(* PLC project Arbeitsmaschine7, KW-Software MULTIPROG 5.35 *)
(* stored: companyURL www.kw-software.com, productRelease Build 434, creationDateTime 2012-11-13T09:01:25, version 1352793685, modificationDateTime 2012-11-13T09:01:25 *)

(* Layer 3: Ablaufebene --> Greift auf Layer 2 zu. Der FB spiegelt die Funktion "Transport nach x, Bearbeitung" eines Werkstücks wider. Der Unterschied zum FB "Bearbeiten" aus Layer 2 besteht darin, dass der Bearbeitungsablauf neben dem reinen Bearbeiten des Werkstückes auch die Übernahme/Übergabe, das Transportieren des Werkstücks, die Werkzeugauswahl und die Höhenänderung des Werkzeugs umfasst. Die Ansteuerung der drei Transportzustände (nach links, nach rechts und aus) wird durch zwei Variablen (Transport_nach_links, Transport_nach_rechts) realisiert. Die Ansteuerung der 4 Bearbeitungszustände wird über 3 Variablen (Bearbeiten1, Bearbeiten2, Bearbeiten3) realisiert. Im Anfangsschritt findet keine Bearbeitung statt - kein Bearbeiten/Transportieren/Übergeben/Übernehmen/ Werkzeug auswählen/keine Höhenänderung (Motoren aus). Je nach Setzen der Inputvariablen (alternative Verzweigung) wird ein Werkstück von der entsprechenden Seite übernommen. Liefert FB "Übernahme_gabe" das Quittierungssignal, dass erfolgreich übernommen wurde, schaltet die Transition. Damit wird ein Zustand eingenommen, der erstmal alle Motoren stoppt (Wichtig ist, dass der Transportbandmotor gestoppt wird.). Nun wird entsprechend der Inputvariablen die Auwahl des Werkzeuges vorgenommen. Liefert der FB "Werkzeugauswahl" das Quittierungssignal, dass das Werkzeug erfolgreich ausgewählt wurde, dann schaltet die Transition. Nun wird geprüft, ob ein Verfahren des Werkzeuges nötig ist und das Werkzeug gegebenenfalls verfahren werden muss. Wurde das Werkzeug bereits auf die unterste Position verfahren, so ist kein weiteres Verfahren des Werkzeuges nötig. Ebenfalls ist ein Verfahren des Werkzeuges unnötig, wenn kein Werkstück zur Bearbeitung bereitliegt. Nach erfolgreichem Verfahren des Werkzeuges, liefert der FB "Werkzeughoehe" das Quittierungssignal und die Transition schaltet. Nun wird das Werkzeug entsprechend der Inputvariablen bearbeitet. Wenn die Bearbeitung abgeschlossen ist, wird vom FB "Bearbeiten" ein Quittierungssignal gesendet und die Transition schaltet. Nun wird geprüft, ob ein Verfahren des Werkzeuges nötig ist und das Werkzeug gegebenenfalls verfahren werden muss. Befindet sich das Werkzeug bereits auf der höhsten Position, so ist ein erneutes Verfahren des Werkzeugs nicht nötig. Nach erfolgreichem Verfahren des Werkzeuges liefert der FB "Werkzeughoehe" das Quittierungssignal und die Transition schaltet. Nun schaltet die Transition "T_XXX_ein" und das Werkstück wird in die entsprechende Richtung transportiert. Liefert FB "Transportieren" das Quittierungssignal, dass erfolgreich transportiert wurde, schaltet die Transition. Damit wird ein Zustand eingenommen, der alle Motoren stoppt (Wichtig ist, dass der Transportbandmotor gestoppt wird.). Nach Auswertung der Bedingungen, an welcher Seite das Werkstück übergeben werden muss, wird der Zustand eingenommen,der das Werkstück übergibt. Wurde erfolgreich übergeben, so ist der Bearbeitungsablauf abgeschlossen. Dabei wird auch eine Statusvariable gesetzt (TPB_xxx), die den erfolgreichen Bearbeitungsablauf quittiert, sodass die übergeordnete Steuerung weiß, wann der Transportvorgang und der Bearbeitungsvorgang abgeschlossen ist. FB-Schnittstellen: --------------- Eingangsvariablen: - Bearbeiten1 - Bearbeiten2 - Bearbeiten3 - Transport_nach_links - Transport_nach_rechts Ausgangsvariablen: - TPB_links - TPB_rechts Auftretende Warnungen "Instanz 'FB_xxx' mehrfach verwendet!": Hier ein Textauszug aus der Multiprog-Hilfe: "Die Warnung kann auch in einem Code-Arbeitsblatt in AS auftreten, wenn Sie dieselbe Instanz in verschiedenen Aktionen verwendet haben. Wenn nur eine Instanz zu einem Zeitpunkt ausgeführt wird, ist die Warnung für Sie ohne Bedeutung." *)
FUNCTION_BLOCK Transport_zu_x_Bearbeit
  VAR
    FB_Uebergabe : Uebernahme_gabe;
    FB_Uebernahme : Uebernahme_gabe;
    FB_Bearbeiten : Bearbeiten;
    FB_Werkzeugauswahl : Werkzeugauswahl;
    FB_Werkzeughoehe : Werkzeughoehe;
  END_VAR
  VAR_INPUT
    Transport_nach_links : BOOL := FALSE;
    Transport_nach_rechts : BOOL := FALSE;
  END_VAR
  VAR
    Quittierungssignal_links1 : BOOL := FALSE;
    Quittierungssignal_rechts1 : BOOL := FALSE;
    Quittierungssignal_links2 : BOOL := FALSE;
    Quittierungssignal_rechts2 : BOOL := FALSE;
  END_VAR
  VAR_INPUT
    Bearbeiten1 : BOOL := FALSE;
    Bearbeiten2 : BOOL := FALSE;
    Bearbeiten3 : BOOL := FALSE;
  END_VAR
  VAR
    Sensor_Auswahl : BOOL := FALSE;
    links : BOOL := FALSE;
    rechts : BOOL := FALSE;
    Quittierungssignal_Wahl1 : BOOL := FALSE;
    Quittierungssignal_Wahl2 : BOOL := FALSE;
    Quittierungssignal_Wahl3 : BOOL := FALSE;
    Quittierungssignal_ab : BOOL := FALSE;
    Hoehe_0 : BOOL := FALSE;
    Quittierungssignal_WZ1 : BOOL := FALSE;
    Quittierungssignal_WZ2 : BOOL := FALSE;
    Quittierungssignal_WZ3 : BOOL := FALSE;
    Quittierungssignal_auf : BOOL := FALSE;
    Quittierungssignal_links3 : BOOL := FALSE;
    Quittierungssignal_rechts3 : BOOL := FALSE;
    Quittierungssignal_links4 : BOOL := FALSE;
    Quittierungssignal_rechts4 : BOOL := FALSE;
  END_VAR
  VAR_OUTPUT
    TPB_rechts : BOOL := FALSE;
    TPB_links : BOOL := FALSE;
  END_VAR
  VAR
    FB_Werkzeughoehe_auf : Werkzeughoehe;
    FB_Werkzeughoehe_ab : Werkzeughoehe;
    FB_Positionieren : Positionieren;
    Quittierungssignal_Pos_links : BOOL := FALSE;
    Quittierungssignal_Pos_rechts : BOOL := FALSE;
  END_VAR

(* transition T_Uebergeben_r_aus *)
FB_Uebergabe();
Quittierungssignal_rechts4 := FB_Uebergabe.UeG_UeN_rechts;
IF Quittierungssignal_rechts4 = TRUE
	THEN T_Uebergeben_r_aus := TRUE;
	ELSE T_Uebergeben_r_aus := FALSE;
END_IF;
(* transition T_Uebergeben_l_aus *)
FB_Uebergabe();
Quittierungssignal_links4 := FB_Uebergabe.UeG_UeN_links;
IF Quittierungssignal_links4 = TRUE
	THEN T_Uebergeben_l_aus := TRUE;
	ELSE T_Uebergeben_l_aus := FALSE;
END_IF;
(* transition T_Uebergeben_r_ein *)
FB_Uebernahme();
Quittierungssignal_rechts3 := FB_Uebernahme.UeG_UeN_rechts;
IF Quittierungssignal_rechts3 = TRUE
	THEN T_Uebergeben_r_ein := TRUE; 
	ELSE T_Uebergeben_r_ein := FALSE;
END_IF;
(* transition T_Uebergeben_l_ein *)
FB_Uebernahme();
Quittierungssignal_links3 := FB_Uebernahme.UeG_UeN_links;
IF Quittierungssignal_links3 = TRUE 
	THEN T_Uebergeben_l_ein := TRUE; 
	ELSE T_Uebergeben_l_ein := FALSE;
END_IF;
(* transition T_Hoehe_aufwaerts_aus *)
FB_Werkzeughoehe_auf();
Quittierungssignal_auf := FB_Werkzeughoehe_auf.Hoehe_auf;
IF Quittierungssignal_auf = TRUE
	THEN T_Hoehe_aufwaerts_aus := TRUE;
	ELSE T_Hoehe_aufwaerts_aus := FALSE;
END_IF;
(* transition T_keine_Hoehenaenderung2 *)
FB_Werkzeughoehe();
Hoehe_0 := FB_Werkzeughoehe.Position0;
IF Hoehe_0 = TRUE
	THEN T_keine_Hoehenaenderung2 := TRUE; 
	ELSE T_keine_Hoehenaenderung2 := FALSE;
END_IF;
(* transition T_Hoehe_aufwaerts_ein *)
FB_Werkzeughoehe();
Hoehe_0 := FB_Werkzeughoehe.Position0;
IF Hoehe_0 = FALSE
	THEN T_Hoehe_aufwaerts_ein := TRUE; 
	ELSE T_Hoehe_aufwaerts_ein := FALSE;
END_IF;
(* transition T_Werkzeug3_aus *)
FB_Bearbeiten();
Quittierungssignal_WZ3 := FB_Bearbeiten.BA_WZ3;
IF Quittierungssignal_WZ3 = TRUE
	THEN T_Werkzeug3_aus := TRUE;
	ELSE T_Werkzeug3_aus := FALSE;
END_IF;
(* transition T_Werkzeug2_aus *)
FB_Bearbeiten();
Quittierungssignal_WZ2 := FB_Bearbeiten.BA_WZ2;
IF Quittierungssignal_WZ2 = TRUE
	THEN T_Werkzeug2_aus := TRUE;
	ELSE T_Werkzeug2_aus := FALSE; 
END_IF;
(* transition T_Werkzeug1_aus *)
FB_Bearbeiten();
Quittierungssignal_WZ1 := FB_Bearbeiten.BA_WZ1;
IF Quittierungssignal_WZ1 = TRUE
	THEN T_Werkzeug1_aus := TRUE;
	ELSE T_Werkzeug1_aus := FALSE;
END_IF;
(* transition T_Werkzeug3_ein *)
IF Bearbeiten1 = FALSE AND Bearbeiten2 = FALSE AND Bearbeiten3 = TRUE 
	THEN T_Werkzeug3_ein := TRUE;
	ELSE T_Werkzeug3_ein := FALSE; 
END_IF;
(* transition T_Werkzeug2_ein *)
IF Bearbeiten1 = FALSE AND Bearbeiten2 = TRUE AND Bearbeiten3 = FALSE
	THEN T_Werkzeug2_ein := TRUE; 
	ELSE T_Werkzeug2_ein := FALSE;
END_IF;
(* transition T_Werkzeug1_ein *)
IF Bearbeiten1 = TRUE AND Bearbeiten2 = FALSE AND Bearbeiten3 = FALSE 
	THEN T_Werkzeug1_ein := TRUE;
	ELSE T_Werkzeug1_ein := FALSE; 
END_IF;
(* transition T_Hoehe_abwaerts_aus *)
FB_Werkzeughoehe_ab();
Quittierungssignal_ab := FB_Werkzeughoehe_ab.Hoehe_ab;
IF Quittierungssignal_ab = TRUE 
	THEN T_Hoehe_abwaerts_aus := TRUE; 
	ELSE T_Hoehe_abwaerts_aus := FALSE; 
END_IF;
(* transition T_keine_Hoehenaenderung1 *)
FB_Werkzeughoehe();
Hoehe_0 := FB_Werkzeughoehe.Position0;
IF Hoehe_0 = FALSE
	THEN T_keine_Hoehenaenderung1 := TRUE; 
	ELSE T_keine_Hoehenaenderung1 := FALSE; 
END_IF;
(* transition T_Hoehe_abwaerts_ein *)
FB_Werkzeughoehe();
Hoehe_0 := FB_Werkzeughoehe.Position0;
IF Hoehe_0 = TRUE
	THEN T_Hoehe_abwaerts_ein := TRUE; 
	ELSE T_Hoehe_abwaerts_ein := FALSE; 
END_IF;
(* transition T_Auswahl3_aus *)
FB_Werkzeugauswahl();
Quittierungssignal_Wahl3 := FB_Werkzeugauswahl.Wahl_WZ3;
IF Quittierungssignal_Wahl3 = TRUE
	THEN T_Auswahl3_aus := TRUE; 
	ELSE T_Auswahl3_aus := FALSE;
END_IF;
(* transition T_Auswahl2_aus *)
FB_Werkzeugauswahl();
Quittierungssignal_Wahl2 := FB_Werkzeugauswahl.Wahl_WZ2;
IF Quittierungssignal_Wahl2 = TRUE
	THEN T_Auswahl2_aus := TRUE; 
	ELSE T_Auswahl2_aus := FALSE;
END_IF;
(* transition T_keine_Auswahl *)
FB_Werkzeugauswahl();
Sensor_Auswahl := FB_Werkzeugauswahl.Sensor_Wahl;
links := FB_Werkzeugauswahl.Richtung1;
rechts := FB_Werkzeugauswahl.Richtung2;

IF	Bearbeiten1 = TRUE AND
	Bearbeiten2 = FALSE AND
	Bearbeiten3 = FALSE AND
	Sensor_Auswahl = TRUE AND
	links = TRUE AND
	rechts = FALSE
OR	Bearbeiten1 = FALSE AND
	Bearbeiten2 = TRUE AND
	Bearbeiten3 = FALSE AND
	Sensor_Auswahl = FALSE AND
	links = FALSE AND 
	rechts = FALSE 
OR 	Bearbeiten1 = FALSE AND
	Bearbeiten2 = FALSE AND
	Bearbeiten3 = TRUE AND
	Sensor_Auswahl = TRUE AND
	links = FALSE AND
	rechts = TRUE 
THEN T_keine_Auswahl := TRUE; 
ELSE T_keine_Auswahl := FALSE; 
END_IF;
(* transition T_Auswahl1_aus *)
FB_Werkzeugauswahl();
Quittierungssignal_Wahl1 := FB_Werkzeugauswahl.Wahl_WZ1;
IF Quittierungssignal_Wahl1 = TRUE
	THEN T_Auswahl1_aus := TRUE; 
	ELSE T_Auswahl1_aus := FALSE;
END_IF;
(* transition T_Auswahl3_ein *)
IF Bearbeiten1 = FALSE AND Bearbeiten2 = FALSE AND Bearbeiten3 = TRUE
	THEN T_Auswahl3_ein := TRUE;
	ELSE T_Auswahl3_ein := FALSE;
END_IF;
(* transition T_Auswahl2_ein *)
IF Bearbeiten1 = FALSE AND Bearbeiten2 = TRUE AND Bearbeiten3 = FALSE 
	THEN T_Auswahl2_ein := TRUE;
	ELSE T_Auswahl2_ein := FALSE;
END_IF;
(* transition T_Auswahl1_ein *)
IF Bearbeiten1 = TRUE AND Bearbeiten2 = FALSE AND Bearbeiten3 = FALSE 
	THEN T_Auswahl1_ein := TRUE;
	ELSE T_Auswahl1_ein := FALSE;
END_IF;
(* transition T_Uebernehmen_r_aus *)
FB_Uebernahme();
Quittierungssignal_rechts1 := FB_Uebernahme.UeG_UeN_rechts;
IF Quittierungssignal_rechts1 = TRUE
	THEN T_Uebernehmen_r_aus := TRUE; 
	ELSE T_Uebernehmen_r_aus := FALSE;
END_IF;
(* transition T_Uebernehmen_l_aus *)
FB_Uebernahme();
Quittierungssignal_links1 := FB_Uebernahme.UeG_UeN_links;
IF Quittierungssignal_links1 = TRUE
	THEN T_Uebernehmen_l_aus := TRUE;
	ELSE T_Uebernehmen_l_aus := FALSE;
END_IF;
(* transition T_Uebernehmen_r_ein *)
IF Transport_nach_links = FALSE AND Transport_nach_rechts = TRUE
	THEN T_Uebernehmen_r_ein := TRUE; 
	ELSE T_Uebernehmen_r_ein := FALSE;
END_IF;
(* transition T_Uebernehmen_l_ein *)
IF Transport_nach_links = TRUE AND Transport_nach_rechts = FALSE 
	THEN T_Uebernehmen_l_ein := TRUE;
	ELSE T_Uebernehmen_l_ein := FALSE;
END_IF;
(* transition T_Positionieren_l_ein *)
IF Bearbeiten1 = FALSE AND Bearbeiten2 = FALSE AND Bearbeiten3 = TRUE 
	THEN T_Positionieren_l_ein := TRUE;
	ELSE T_Positionieren_l_ein := FALSE;
END_IF;
(* transition T_Positionieren_r_ein *)
IF Bearbeiten1 = TRUE AND Bearbeiten2 = FALSE AND Bearbeiten3 = FALSE 
	THEN T_Positionieren_r_ein := TRUE; 
	ELSE T_Positionieren_r_ein := FALSE;
END_IF;
(* transition T_kein_Positionieren *)
IF Bearbeiten1 = FALSE AND Bearbeiten2 = TRUE AND Bearbeiten3 = FALSE
	THEN T_kein_Positionieren := TRUE; 
	ELSE T_kein_Positionieren := FALSE; 
END_IF; 
(* transition T_Positionieren_l_aus *)
FB_Positionieren(); 
Quittierungssignal_Pos_links := FB_Positionieren.Pos_links;

IF Quittierungssignal_Pos_links = TRUE
	THEN T_Positionieren_l_aus := TRUE;
	ELSE T_Positionieren_l_aus := FALSE; 
END_IF;
(* transition T_Positionieren_r_aus *)
FB_Positionieren(); 
Quittierungssignal_Pos_rechts := FB_Positionieren.Pos_rechts;

IF Quittierungssignal_Pos_rechts = TRUE
	THEN T_Positionieren_r_aus := TRUE;
	ELSE T_Positionieren_r_aus := FALSE; 
END_IF;
INITIAL_STEP Motor_aus0:
END_STEP
TRANSITION FROM Motor_aus0 TO Motor_links
  := T_Uebernehmen_l_ein;
END_TRANSITION
TRANSITION FROM Motor_aus0 TO Motor_rechts
  := T_Uebernehmen_r_ein;
END_TRANSITION
STEP Motor_links:
END_STEP
TRANSITION FROM Motor_links TO Motor_aus
  := T_Uebernehmen_l_aus;
END_TRANSITION
STEP Motor_rechts:
END_STEP
TRANSITION FROM Motor_rechts TO Motor_aus
  := T_Uebernehmen_r_aus;
END_TRANSITION
STEP Motor_aus:
END_STEP
TRANSITION FROM Motor_aus TO Motor_Auswahl_links
  := T_Auswahl1_ein;
END_TRANSITION
TRANSITION FROM Motor_aus TO Motor_Auswahl_aus
  := T_Auswahl2_ein;
END_TRANSITION
TRANSITION FROM Motor_aus TO Motor_Auswahl_rechts
  := T_Auswahl3_ein;
END_TRANSITION
TRANSITION FROM Motor_aus TO Motor_Auswahl_aus2
  := T_keine_Auswahl;
END_TRANSITION
STEP Motor_Auswahl_links:
END_STEP
TRANSITION FROM Motor_Auswahl_links TO Motor_Auswahl_aus2
  := T_Auswahl1_aus;
END_TRANSITION
STEP Motor_Auswahl_aus:
END_STEP
TRANSITION FROM Motor_Auswahl_aus TO Motor_Auswahl_aus2
  := T_Auswahl2_aus;
END_TRANSITION
STEP Motor_Auswahl_rechts:
END_STEP
TRANSITION FROM Motor_Auswahl_rechts TO Motor_Auswahl_aus2
  := T_Auswahl3_aus;
END_TRANSITION
STEP Motor_Auswahl_aus2:
END_STEP
TRANSITION FROM Motor_Auswahl_aus2 TO Motor_Hoehe_rechts
  := T_Hoehe_abwaerts_ein;
END_TRANSITION
TRANSITION FROM Motor_Auswahl_aus2 TO Motor_Hoehe_aus
  := T_keine_Hoehenaenderung1;
END_TRANSITION
STEP Motor_Hoehe_rechts:
END_STEP
TRANSITION FROM Motor_Hoehe_rechts TO Motor_Hoehe_aus
  := T_Hoehe_abwaerts_aus;
END_TRANSITION
STEP Motor_Hoehe_aus:
END_STEP
TRANSITION FROM Motor_Hoehe_aus TO Motor_Bearbeiten1
  := T_Werkzeug1_ein;
END_TRANSITION
TRANSITION FROM Motor_Hoehe_aus TO Motor_Bearbeiten2
  := T_Werkzeug2_ein;
END_TRANSITION
TRANSITION FROM Motor_Hoehe_aus TO Motor_Bearbeiten3
  := T_Werkzeug3_ein;
END_TRANSITION
STEP Motor_Bearbeiten1:
END_STEP
TRANSITION FROM Motor_Bearbeiten1 TO Motor_Bearbeiten_aus
  := T_Werkzeug1_aus;
END_TRANSITION
STEP Motor_Bearbeiten2:
END_STEP
TRANSITION FROM Motor_Bearbeiten2 TO Motor_Bearbeiten_aus
  := T_Werkzeug2_aus;
END_TRANSITION
STEP Motor_Bearbeiten3:
END_STEP
TRANSITION FROM Motor_Bearbeiten3 TO Motor_Bearbeiten_aus
  := T_Werkzeug3_aus;
END_TRANSITION
STEP Motor_Bearbeiten_aus:
END_STEP
TRANSITION FROM Motor_Bearbeiten_aus TO Motor_Hoehe_links
  := T_Hoehe_aufwaerts_ein;
END_TRANSITION
TRANSITION FROM Motor_Bearbeiten_aus TO Motor_Hoehe_aus2
  := T_keine_Hoehenaenderung2;
END_TRANSITION
STEP Motor_Hoehe_links:
END_STEP
TRANSITION FROM Motor_Hoehe_links TO Motor_Hoehe_aus2
  := T_Hoehe_aufwaerts_aus;
END_TRANSITION
STEP Motor_Hoehe_aus2:
END_STEP
TRANSITION FROM Motor_Hoehe_aus2 TO Motor_Auswahl_links2
  := T_Positionieren_l_ein;
END_TRANSITION
TRANSITION FROM Motor_Hoehe_aus2 TO Motor_Auswahl_rechts2
  := T_Positionieren_r_ein;
END_TRANSITION
TRANSITION FROM Motor_Hoehe_aus2 TO Motor_Auswahl_aus3
  := T_kein_Positionieren;
END_TRANSITION
STEP Motor_Auswahl_links2:
END_STEP
TRANSITION FROM Motor_Auswahl_links2 TO Motor_Auswahl_aus3
  := T_Positionieren_l_aus;
END_TRANSITION
STEP Motor_Auswahl_rechts2:
END_STEP
TRANSITION FROM Motor_Auswahl_rechts2 TO Motor_Auswahl_aus3
  := T_Positionieren_r_aus;
END_TRANSITION
STEP Motor_Auswahl_aus3:
END_STEP
TRANSITION FROM Motor_Auswahl_aus3 TO Motor_links3
  := T_Uebergeben_l_ein;
END_TRANSITION
TRANSITION FROM Motor_Auswahl_aus3 TO Motor_rechts3
  := T_Uebergeben_r_ein;
END_TRANSITION
STEP Motor_links3:
END_STEP
TRANSITION FROM Motor_links3 TO Quittierung_l
  := T_Uebergeben_l_aus;
END_TRANSITION
STEP Motor_rechts3:
END_STEP
TRANSITION FROM Motor_rechts3 TO Quittierung_r
  := T_Uebergeben_r_aus;
END_TRANSITION
STEP Quittierung_l:
END_STEP
TRANSITION FROM Quittierung_l TO Endschritt_3  (* T_sofort_weiter13 *)
  := TRUE;
END_TRANSITION
STEP Quittierung_r:
END_STEP
TRANSITION FROM Quittierung_r TO Endschritt_3  (* T_sofort_weiter14 *)
  := TRUE;
END_TRANSITION
STEP Endschritt_3:
END_STEP

ACTION Endschritt_Bearbeitung:
FB_Uebergabe ( Uebergeben := FALSE , Uebernehmen := FALSE );
FB_Uebernahme ( Uebergeben := FALSE , Uebernehmen := FALSE ); 
FB_Bearbeiten ( Bearbeitung1 := FALSE , Bearbeitung2 := FALSE , Bearbeitung3 := FALSE );
FB_Werkzeugauswahl ( Werkzeug1 := FALSE , Werkzeug2 := FALSE , Werkzeug3 := FALSE );
FB_Werkzeughoehe ( Hoehe_aufwaerts := FALSE , Hoehe_abwaerts := FALSE ); 
FB_Positionieren ( Positionierung_links := FALSE , Positionierung_rechts := FALSE );
END_ACTION

ACTION Quittierung_rechts3:
TPB_rechts := TRUE;
END_ACTION

ACTION Quittierung_links3:
TPB_links := TRUE;
END_ACTION

ACTION Uebergeben_rechts:
FB_Uebergabe ( Richtung := TRUE , Uebergeben := TRUE , Uebernehmen := FALSE );
END_ACTION

ACTION Uebergeben_links:
FB_Uebergabe ( Richtung := FALSE , Uebergeben := TRUE , Uebernehmen := FALSE );
END_ACTION

ACTION Hoehe_aufwaerts:
FB_Werkzeughoehe_auf ( Hoehe_aufwaerts := TRUE , Hoehe_abwaerts := FALSE );
END_ACTION

ACTION Bearbeiten_aus:
FB_Bearbeiten ( Bearbeitung1 := FALSE , Bearbeitung2 := FALSE , Bearbeitung3 := FALSE );
END_ACTION

ACTION Bearbeitung3:
FB_Bearbeiten ( Bearbeitung1 := FALSE , Bearbeitung2 := FALSE , Bearbeitung3 := TRUE);
END_ACTION

ACTION Bearbeitung2:
FB_Bearbeiten ( Bearbeitung1 := FALSE , Bearbeitung2 := TRUE , Bearbeitung3 := FALSE );
END_ACTION

ACTION Bearbeitung1:
FB_Bearbeiten ( Bearbeitung1 := TRUE , Bearbeitung2 := FALSE , Bearbeitung3 := FALSE );
END_ACTION

ACTION Hoehenaenderung_aus:
FB_Werkzeughoehe_auf ( Hoehe_aufwaerts := FALSE , Hoehe_abwaerts := FALSE );
FB_Werkzeughoehe_ab ( Hoehe_aufwaerts := FALSE , Hoehe_abwaerts := FALSE );
END_ACTION

ACTION Hoehe_abwaerts:
FB_Werkzeughoehe_ab ( Hoehe_abwaerts := TRUE , Hoehe_aufwaerts := FALSE );
END_ACTION

ACTION Auswahl_aus:
FB_Werkzeugauswahl ( Werkzeug1 := FALSE , Werkzeug2 := FALSE , Werkzeug3 := FALSE );
END_ACTION

ACTION Auswahl_WZ3:
FB_Werkzeugauswahl ( Werkzeug1 := FALSE , Werkzeug2 := FALSE , Werkzeug3 := TRUE );
END_ACTION

ACTION Auswahl_WZ2:
FB_Werkzeugauswahl ( Werkzeug1 := FALSE , Werkzeug2 := TRUE , Werkzeug3 := FALSE );
END_ACTION

ACTION Auswahl_WZ1:
FB_Werkzeugauswahl ( Werkzeug1 := TRUE , Werkzeug2 := FALSE , Werkzeug3 := FALSE );
END_ACTION

ACTION Uebernehmen_aus:
FB_Transportieren ( Transportieren_links := FALSE , Transportieren_rechts := FALSE );
FB_Uebergabe ( Uebergeben := FALSE , Uebernehmen := FALSE );
FB_Uebernahme ( Uebergeben := FALSE , Uebernehmen := FALSE );
END_ACTION

ACTION Uebernehmen_rechts:
FB_Uebernahme ( Richtung := FALSE , Uebergeben := FALSE , Uebernehmen := TRUE );
END_ACTION

ACTION Uebernehmen_links:
FB_Uebernahme ( Richtung := TRUE , Uebergeben := FALSE , Uebernehmen := TRUE );
END_ACTION

ACTION Bearbeitung_aus:
FB_Uebergabe ( Uebergeben := FALSE , Uebernehmen := FALSE );
FB_Uebernahme ( Uebergeben := FALSE , Uebernehmen := FALSE ); 
FB_Bearbeiten ( Bearbeitung1 := FALSE , Bearbeitung2 := FALSE , Bearbeitung3 := FALSE );
FB_Werkzeugauswahl ( Werkzeug1 := FALSE , Werkzeug2 := FALSE , Werkzeug3 := FALSE );
FB_Werkzeughoehe ( Hoehe_aufwaerts := FALSE , Hoehe_abwaerts := FALSE ); 
FB_Positionieren ( Positionierung_links := FALSE , Positionierung_rechts := FALSE );
END_ACTION

ACTION Positionieren_aus:
FB_Positionieren( Positionierung_links := FALSE , Positionierung_rechts := FALSE );
END_ACTION

ACTION Positionieren_rechts:
FB_Positionieren ( Positionierung_links := FALSE , Positionierung_rechts := TRUE );
END_ACTION

ACTION Positionieren_links:
FB_Positionieren ( Positionierung_links := TRUE , Positionierung_rechts := FALSE );
END_ACTION
END_FUNCTION_BLOCK
